{attribute 'linkalways'} 
{attribute 'no_explicit_call' := 'This FB is a CLASS and must be accessed using methods or properties'}
{attribute 'enable_dynamic_creation'}
FUNCTION_BLOCK Node_F_VN_GetNumberOfElements EXTENDS VisionNode
VAR
    ipContainer : _ITcVnContainer;
    nNumberOfElements : _ULINT(0);
    hrPrev : _HRESULT(S_OK);
	hresult : _HRESULT(S_OK);
END_VAR

METHOD PUBLIC  Clone : I_Node
VAR
	pNode : POINTER TO Node_F_VN_GetNumberOfElements;
END_VAR
pNode := __NEW(Node_F_VN_GetNumberOfElements);
Clone := pNode^;
END_METHOD

METHOD FB_init : BOOL
VAR_INPUT
	bInitRetains : BOOL; // if TRUE, the retain variables are initialized (warm start / cold start)
	bInCopyCode : BOOL;  // if TRUE, the instance afterwards gets moved into the copy code (online change)
END_VAR
AddInput('ipContainer', ipContainer);
AddInput('hrPrev', hrPrev);
AddOutput('nNumberOfElements', nNumberOfElements);
AddOutput('hresult',hresult);
END_METHOD

METHOD PROTECTED OnExecute : HRESULT
hresult.Value := F_VN_GetNumberOfElements(
	ipContainer := ipContainer.Value,
    nNumberOfElements := nNumberOfElements.Value,
	hrPrev:= hrPrev.Value);
END_METHOD

METHOD PUBLIC PreExecutionCheck
VAR_INPUT
	Check : I_PreExecutionChecks;
END_VAR
Check.IsTrue(ipContainer.IsValid, 'ipContainer must be a valid container');
END_METHOD

END_FUNCTION_BLOCK

(* stored: Version 1.1.0.1, ProductVersion 3.1.4024.13
   POU Node_F_VN_GetNumberOfElements: Id {e8d23201-3ff4-0097-0d97-1347e940ef78}, SpecialFunc None
   Folder Constructor: Id {219b0797-48fc-0f3a-1ef2-61408f31ffef}
   Method Clone: Id {8057b64e-d3b9-02f2-2319-cb2b27d55081}
   Method FB_init: Id {833dfecf-501b-0b2a-0dda-6e53bd079620}
   Method OnExecute: Id {6a054dd5-115e-0803-1bdd-ba718ae30def}
   Method PreExecutionCheck: Id {71474760-06f5-01e6-2b81-67fbbe9cbcc7} *)
